FUNCTION FUN_AX8000_GetMotorTemperatureUDINT : UDINT
VAR_INPUT
		Axis									:	Tc2_Mc2.AXIS_REF;
		Channel									:	STRING;
END_VAR
VAR
		CoERead 								:	Tc2_Mc2_Drive.FB_CoERead;
		CoEReadValue 							:	UDINT;
		Busy									:	BOOL;
END_VAR

// AX8000 Get Motor Temperature
// This block is made for inspirational purposes.
// Please make your own version that complies with your / your company´s programming vision
// Version 1.0 - Initial Version
//-----------------------------------------------------------------------------------------

IF NOT CoERead.Busy AND busy THEN
	IF NOT CoERead.error THEN
		FUN_AX8000_GetMotorTemperatureUDINT := CoEReadValue;
	END_IF
END_IF
CoERead(Axis:=Axis,NetId:='',pDstBuf:=ADR(CoEReadValue),BufLen:=SIZEOF(CoEReadValue));
IF Channel = 'A' THEN
	CoERead.Index := 16#32C1; 
END_IF
IF Channel = 'B' THEN
	CoERead.Index := 16#36C1; 
END_IF
CoERead.SubIndex := 0 ;
CoERead.Execute := TRUE;
IF CoERead.Busy THEN
	Busy :=1;
END_IF

END_FUNCTION

(* stored: Version 1.1.0.1, ProductVersion 3.1.4024.14
   POU FUN_AX8000_GetMotorTemperatureUDINT: Id {8d4dd7cf-77da-430b-a4c1-22d6e5e2bae3}, SpecialFunc None *)
